FUNCTION_BLOCK TrafficLightController
VAR_INPUT
	buttonPressed : BOOL;  // Pedestrian button pressed
	vehicleDetected : BOOL;  // Vehicle detected
	emergencyVehicleDetected : BOOL;  // Emergency vehicle detected
END_VAR

VAR_OUTPUT
	greenLight : BOOL;
	yellowLight : BOOL;
	redLight : BOOL;
END_VAR

VAR
	state : INT := 0;  // Current state variable
	prevState : INT := -1;  // Previous state variable (initialized to an invalid state)
	greenTimer : TIME := T#0s;  // Timer for green light duration
	yellowTimer : TIME := T#0s;  // Timer for yellow light duration
	redTimer : TIME := T#0s;  // Timer for red light duration
	pedestrianTimer : TIME := T#0s;  // Timer for pedestrian light duration
	emergencyTimer : TIME := T#0s;  // Timer for emergency vehicle passage
	currentTimer : TIME := T#0s;  // General timer variable for state timing
END_VAR

BEGIN
	// State machine logic
	CASE state OF
		0:  // State 0: Initialize
			greenLight := FALSE;
			yellowLight := FALSE;
			redLight := FALSE;
			IF emergencyVehicleDetected THEN
				state := 5;  // to State 5: Emergency Vehicle
			ELSIF buttonPressed THEN
				state := 4;  // to State 4: Pedestrian Wait
			ELSIF vehicleDetected THEN
				state := 1;  // to State 1: Green Light
			END_IF;

		1:  // State 1: Green Light
			greenLight := TRUE;
			yellowLight := FALSE;
			redLight := FALSE;
			IF vehicleDetected OR (T_PLC_MS() - greenTimer >= T#10s) THEN
				state := 2;  // to State 2: Yellow Light
				yellowTimer := T_PLC_MS();
			END_IF;

		2:  // State 2: Yellow Light
			greenLight := FALSE;
			yellowLight := TRUE;
			redLight := FALSE;
			IF (T_PLC_MS() - yellowTimer >= T#5s) THEN
				state := 3;  // to State 3: Red Light
				redTimer := T_PLC_MS();
			END_IF;

		3:  // State 3: Red Light
			greenLight := FALSE;
			yellowLight := FALSE;
			redLight := TRUE;
			IF (T_PLC_MS() - redTimer >= T#15s) THEN
				IF buttonPressed THEN
					state := 4;  // to State 4: Pedestrian Wait
					pedestrianTimer := T_PLC_MS();
				ELSIF emergencyVehicleDetected THEN
					state := 5;  // to State 5: Emergency Vehicle
					emergencyTimer := T_PLC_MS();
				ELSE
					state := 1;  // back to State 1: Green Light
					greenTimer := T_PLC_MS();
				END_IF;
			END_IF;

		4:  // State 4: Pedestrian Wait
			greenLight := FALSE;
			yellowLight := FALSE;
			redLight := TRUE;
			IF (T_PLC_MS() - pedestrianTimer >= T#10s) THEN
				state := 3;  // back to State 3: Red Light
				redTimer := T_PLC_MS();
			END_IF;

		5:  // State 5: Emergency Vehicle
			greenLight := FALSE;
			yellowLight := TRUE;
			redLight := FALSE;
			IF (T_PLC_MS() - emergencyTimer >= T#10s) THEN
				state := 3;  // back to State 3: Red Light
				redTimer := T_PLC_MS();
			END_IF;
	END_CASE;
END_FUNCTION_BLOCK